SUBAPPLICATION Uebung_002b2 (* DigitalInput_I1/_I2/_I3 auf DigitalOutput_Q1 *)
  (* Standard: 61499-2; Description: Copyright (c) 2023 Meisterschulen am Ostbahnhof This program and the accompanying materials are made available under the terms of the Eclipse Public License 2.0 which is available at https://www.eclipse.org/legal/epl-2.0/ SPDX-License-Identifier: EPL-2.0 *)
  (* Version 1.0, 2023-10-23, Franz Höpfinger, Meisterschulen am Ostbahnhof *)
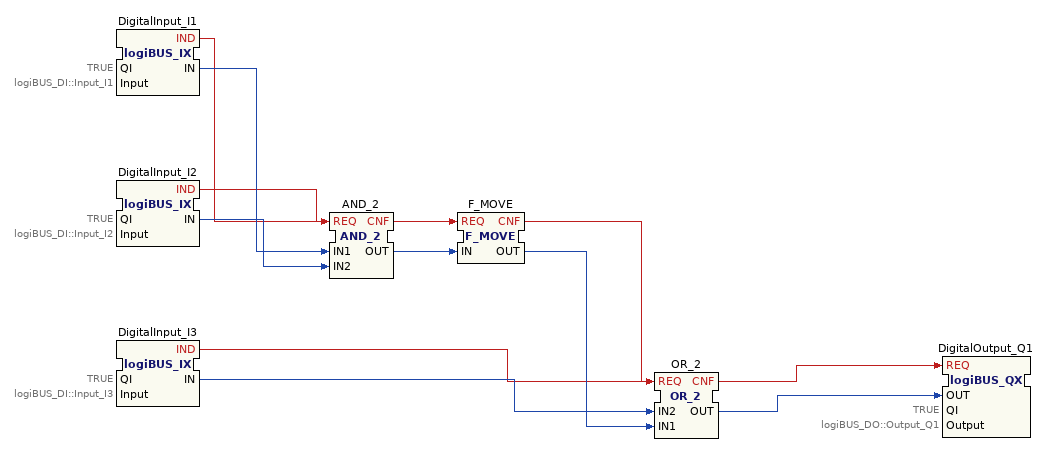
  FBS
    DigitalOutput_Q1 : logiBUS_QX(QI := TRUE, Output := logiBUS_DO::Output_Q1);
    DigitalInput_I1 : logiBUS_IX(QI := TRUE, Input := logiBUS_DI::Input_I1);
    DigitalInput_I2 : logiBUS_IX(QI := TRUE, Input := logiBUS_DI::Input_I2);
    AND_2 : iec61131::bitwiseOperators::AND_2;
    DigitalInput_I3 : logiBUS_IX(QI := TRUE, Input := logiBUS_DI::Input_I3);
    OR_2 : iec61131::bitwiseOperators::OR_2;
    F_MOVE : iec61131::arithmetic::F_MOVE; {SET_ATTRIBUTE(DataType, BOOL)} {SET_ATTRIBUTE(DataType, BOOL)}
  END_FBS
  EVENT_CONNECTIONS
    DigitalInput_I1.IND TO AND_2.REQ;
    DigitalInput_I2.IND TO AND_2.REQ;
    OR_2.CNF TO DigitalOutput_Q1.REQ;
    DigitalInput_I3.IND TO OR_2.REQ;
    F_MOVE.CNF TO OR_2.REQ;
    AND_2.CNF TO F_MOVE.REQ;
  END_CONNECTIONS
  DATA_CONNECTIONS
    DigitalInput_I1.IN TO AND_2.IN1;
    DigitalInput_I2.IN TO AND_2.IN2;
    DigitalInput_I3.IN TO OR_2.IN2;
    OR_2.OUT TO DigitalOutput_Q1.OUT;
    F_MOVE.OUT TO OR_2.IN1;
    AND_2.OUT TO F_MOVE.IN;
  END_CONNECTIONS
END_SUBAPPLICATION
